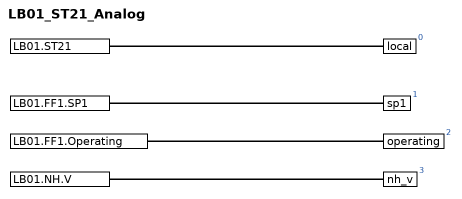
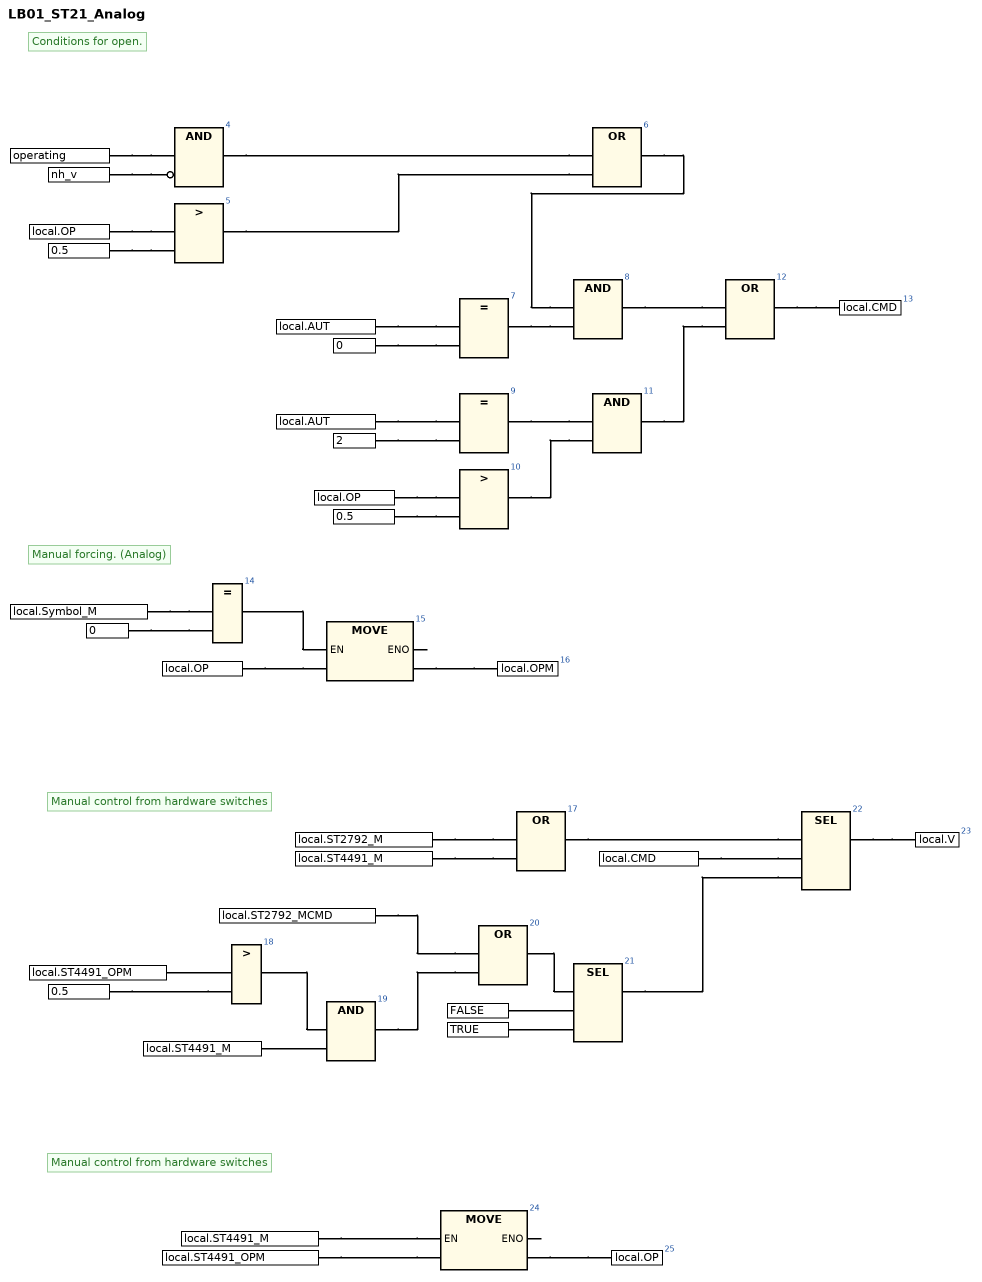
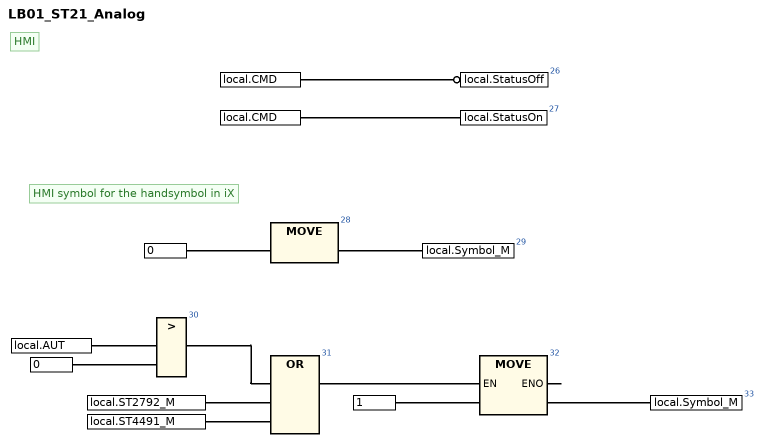
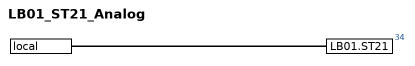
local := LB01.ST21;
sp1 := LB01.FF1.SP1;
operating := LB01.FF1.Operating;
nh_v := LB01.NH.V;
// Conditions for open.
local.CMD := (operating AND NOT nh_v OR local.OP > 0.5) AND local.AUT = 0 OR local.AUT = 2 AND local.OP > 0.5;
// Manual forcing. (Analog)
IF local.Symbol_M = 0 THEN _w1 := local.OP; END_IF
local.OPM := _w1;
// Manual control from hardware switches
local.V := SEL(local.ST2792_M OR local.ST4491_M, local.CMD, SEL(local.ST2792_MCMD OR local.ST4491_OPM > 0.5 AND local.ST4491_M, FALSE, TRUE));
// Manual control from hardware switches
IF local.ST4491_M THEN _w2 := local.ST4491_OPM; END_IF
local.OP := _w2;
// HMI
local.StatusOff := NOT local.CMD;
local.StatusOn := local.CMD;
// HMI symbol for the handsymbol in iX
local.Symbol_M := 0;
IF local.AUT > 0 OR local.ST2792_M OR local.ST4491_M THEN _w3 := 1; END_IF
local.Symbol_M := _w3;
LB01.ST21 := local;

END_PROGRAM

// Device/AREA1/B001/LB01/Fan/TF1/LB01_TF1_OneSpeed
PROGRAM LB01_TF1_OneSpeed
VAR
	local:strFan_Onespeed;
	_BE_Fan2:_BE_Fan_2;
	AlarmFbAl01: _BE_AlarmAckRequired;
	AlarmFbAl02: _BE_AlarmAckRequired;
	fb_OperationalTime: _BE_OperationalTime;
	ackAl01: BOOL;
	ackAl02: BOOL;
	fanGuardOk: BOOL;
END_VAR

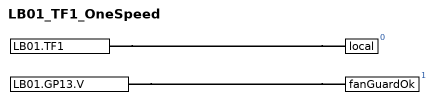
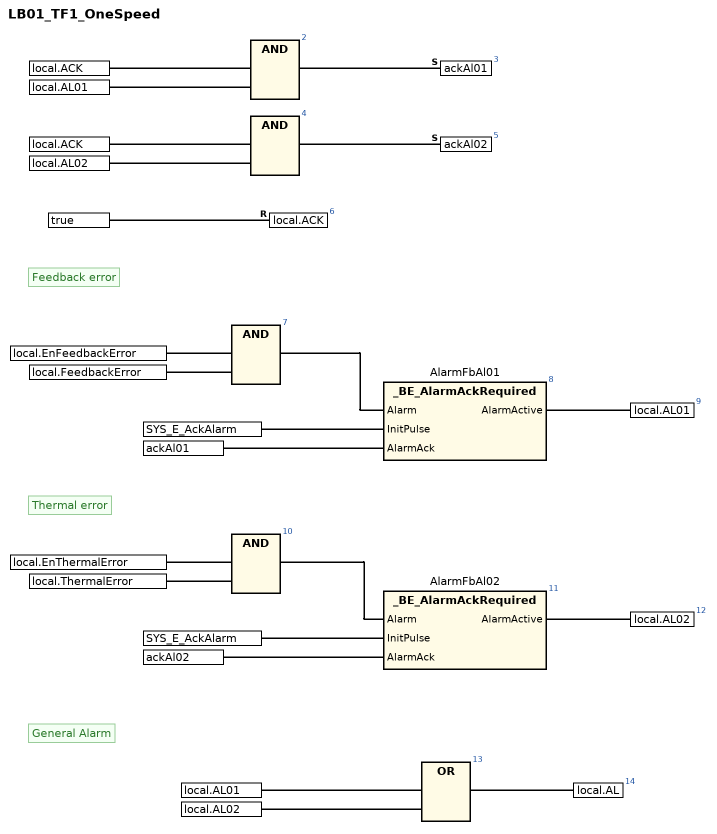
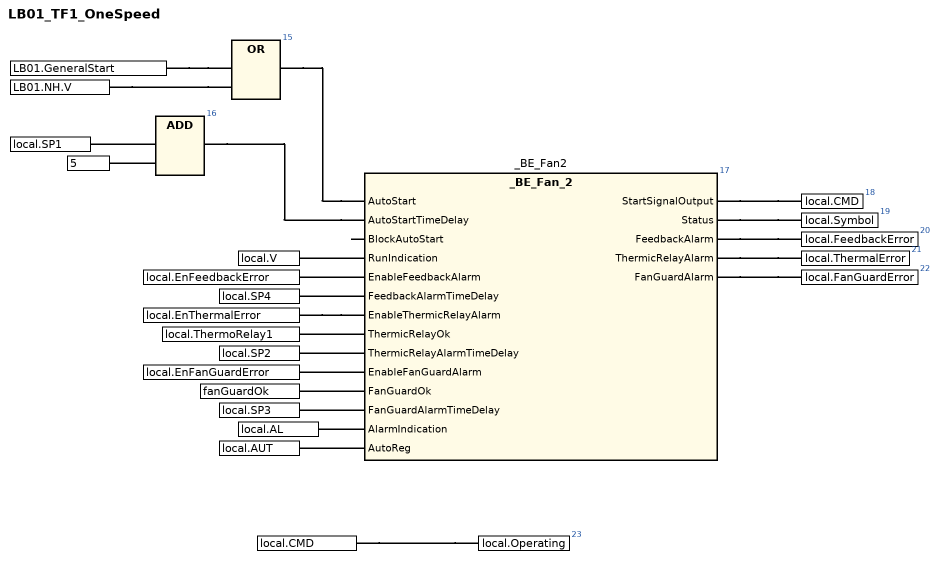
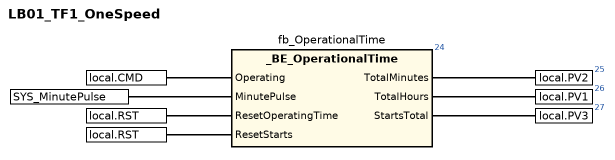
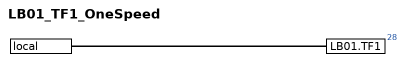
local := LB01.TF1;
fanGuardOk := LB01.GP13.V;
ackAl01 S= local.ACK AND local.AL01;
ackAl02 S= local.ACK AND local.AL02;
local.ACK R= true;
// Feedback error
AlarmFbAl01(
    Alarm := local.EnFeedbackError AND local.FeedbackError,
    InitPulse := SYS_E_AckAlarm,
    AlarmAck := ackAl01); // _BE_AlarmAckRequired
local.AL01 := AlarmFbAl01.AlarmActive;
// Thermal error
AlarmFbAl02(
    Alarm := local.EnThermalError AND local.ThermalError,
    InitPulse := SYS_E_AckAlarm,
    AlarmAck := ackAl02); // _BE_AlarmAckRequired
local.AL02 := AlarmFbAl02.AlarmActive;
// General Alarm
local.AL := local.AL01 OR local.AL02;
_BE_Fan2(
    AutoStart := LB01.GeneralStart OR LB01.NH.V,
    AutoStartTimeDelay := local.SP1 + 5,
    RunIndication := local.V,
    EnableFeedbackAlarm := local.EnFeedbackError,
    FeedbackAlarmTimeDelay := local.SP4,
    EnableThermicRelayAlarm := local.EnThermalError,
    ThermicRelayOk := local.ThermoRelay1,
    ThermicRelayAlarmTimeDelay := local.SP2,
    EnableFanGuardAlarm := local.EnFanGuardError,
    FanGuardOk := fanGuardOk,
    FanGuardAlarmTimeDelay := local.SP3,
    AlarmIndication := local.AL,
    AutoReg := local.AUT); // _BE_Fan_2
local.CMD := _BE_Fan2.StartSignalOutput;
local.Symbol := _BE_Fan2.Status;
local.FeedbackError := _BE_Fan2.FeedbackAlarm;
local.ThermalError := _BE_Fan2.ThermicRelayAlarm;
local.FanGuardError := _BE_Fan2.FanGuardAlarm;
local.Operating := local.CMD;
fb_OperationalTime(
    Operating := local.CMD,
    MinutePulse := SYS_MinutePulse,
    ResetOperatingTime := local.RST,
    ResetStarts := local.RST); // _BE_OperationalTime
local.PV2 := fb_OperationalTime.TotalMinutes;
local.PV1 := fb_OperationalTime.TotalHours;
local.PV3 := fb_OperationalTime.StartsTotal;
LB01.TF1 := local;

END_PROGRAM

// Device/AREA1/B001/LB01/Fan/TF1/LB01_TF1_TwoSpeed
PROGRAM LB01_TF1_TwoSpeed
VAR
	local:strFan_TwoSpeed;
	ControlTwoSpeed: _BE_FanTwoSpeed;
	AlarmFbAl03: _BE_AlarmAckRequired;
	AlarmFbAl04: _BE_AlarmAckRequired;
	AlarmFbAl05: _BE_AlarmAckRequired;
	AlarmFbAl06: _BE_AlarmAckRequired;
	ackAl03: BOOL;
	ackAl04: BOOL;
	ackAl05: BOOL;
	ackAl06: BOOL;
	fb_OperationalTime: _BE_OperationalTime;
	localV1: BOOL;
	localthermoRelay2: BOOL;
	fanGuardOk: BOOL;
END_VAR
VAR // added by the converter: edge detectors and wires of the graphical bodies
    _w1 : ANY;
END_VAR

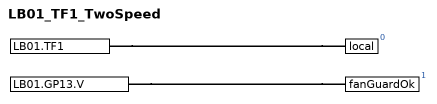
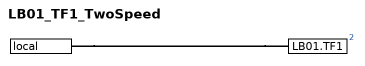
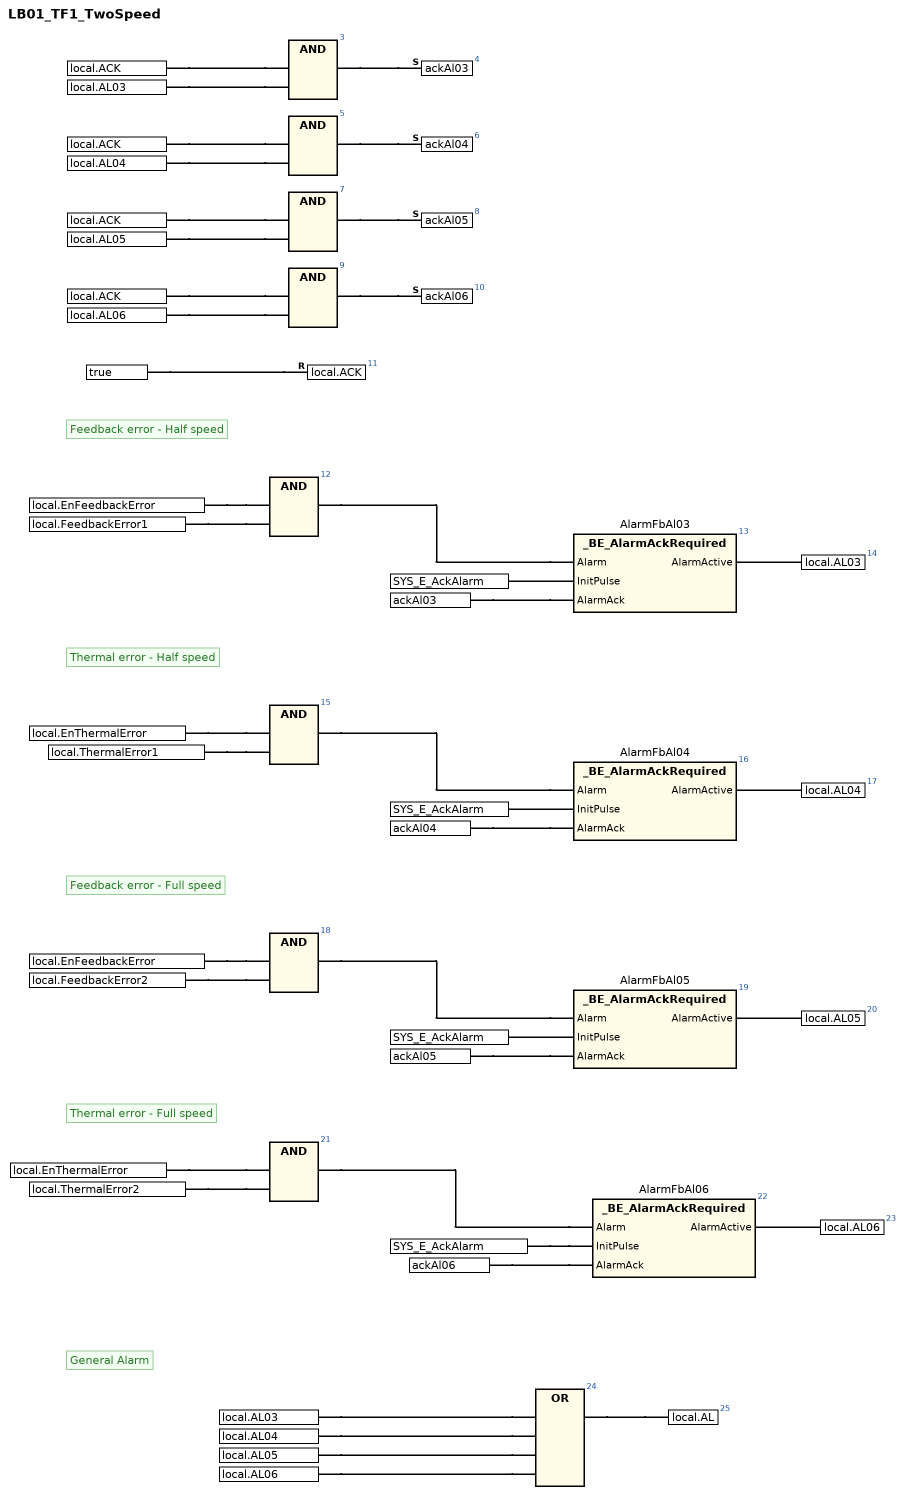
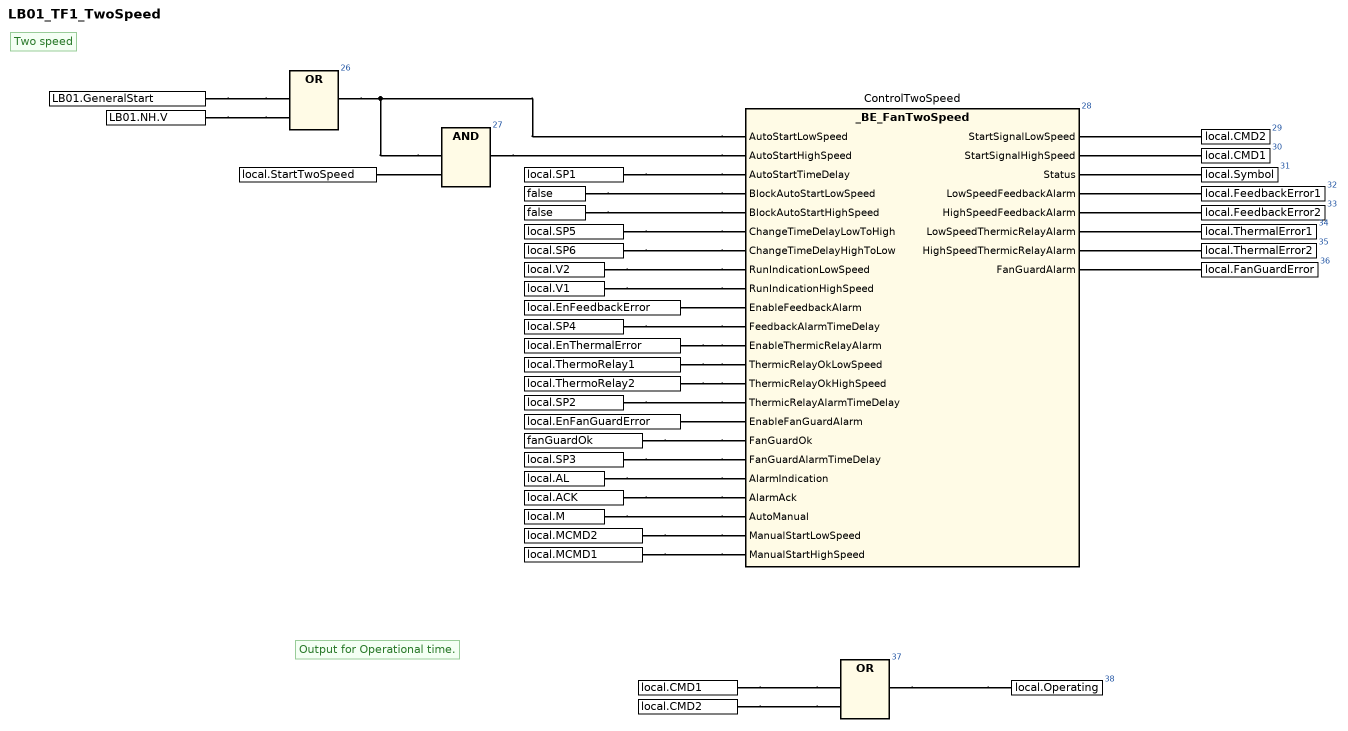
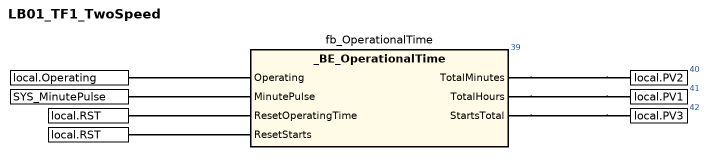
local := LB01.TF1;
fanGuardOk := LB01.GP13.V;
LB01.TF1 := local;
ackAl03 S= local.ACK AND local.AL03;
ackAl04 S= local.ACK AND local.AL04;
ackAl05 S= local.ACK AND local.AL05;
ackAl06 S= local.ACK AND local.AL06;
local.ACK R= true;
// Feedback error - Half speed
AlarmFbAl03(
    Alarm := local.EnFeedbackError AND local.FeedbackError1,
    InitPulse := SYS_E_AckAlarm,
    AlarmAck := ackAl03); // _BE_AlarmAckRequired
local.AL03 := AlarmFbAl03.AlarmActive;
// Thermal error - Half speed
AlarmFbAl04(
    Alarm := local.EnThermalError AND local.ThermalError1,
    InitPulse := SYS_E_AckAlarm,
    AlarmAck := ackAl04); // _BE_AlarmAckRequired
local.AL04 := AlarmFbAl04.AlarmActive;
// Feedback error - Full speed
AlarmFbAl05(
    Alarm := local.EnFeedbackError AND local.FeedbackError2,
    InitPulse := SYS_E_AckAlarm,
    AlarmAck := ackAl05); // _BE_AlarmAckRequired
local.AL05 := AlarmFbAl05.AlarmActive;
// Thermal error - Full speed
AlarmFbAl06(
    Alarm := local.EnThermalError AND local.ThermalError2,
    InitPulse := SYS_E_AckAlarm,
    AlarmAck := ackAl06); // _BE_AlarmAckRequired
local.AL06 := AlarmFbAl06.AlarmActive;
// General Alarm
local.AL := local.AL03 OR local.AL04 OR local.AL05 OR local.AL06;
// Two speed
_w1 := LB01.GeneralStart OR LB01.NH.V;
ControlTwoSpeed(
    AutoStartLowSpeed := _w1,
    AutoStartHighSpeed := _w1 AND local.StartTwoSpeed,
    AutoStartTimeDelay := local.SP1,
    BlockAutoStartLowSpeed := false,
    BlockAutoStartHighSpeed := false,
    ChangeTimeDelayLowToHigh := local.SP5,
    ChangeTimeDelayHighToLow := local.SP6,
    RunIndicationLowSpeed := local.V2,
    RunIndicationHighSpeed := local.V1,
    EnableFeedbackAlarm := local.EnFeedbackError,
    FeedbackAlarmTimeDelay := local.SP4,
    EnableThermicRelayAlarm := local.EnThermalError,
    ThermicRelayOkLowSpeed := local.ThermoRelay1,
    ThermicRelayOkHighSpeed := local.ThermoRelay2,
    ThermicRelayAlarmTimeDelay := local.SP2,
    EnableFanGuardAlarm := local.EnFanGuardError,
    FanGuardOk := fanGuardOk,
    FanGuardAlarmTimeDelay := local.SP3,
    AlarmIndication := local.AL,
    AlarmAck := local.ACK,
    AutoManual := local.M,
    ManualStartLowSpeed := local.MCMD2,
    ManualStartHighSpeed := local.MCMD1); // _BE_FanTwoSpeed
local.CMD2 := ControlTwoSpeed.StartSignalLowSpeed;
local.CMD1 := ControlTwoSpeed.StartSignalHighSpeed;
local.Symbol := ControlTwoSpeed.Status;
local.FeedbackError1 := ControlTwoSpeed.LowSpeedFeedbackAlarm;
local.FeedbackError2 := ControlTwoSpeed.HighSpeedFeedbackAlarm;
local.ThermalError1 := ControlTwoSpeed.LowSpeedThermicRelayAlarm;
local.ThermalError2 := ControlTwoSpeed.HighSpeedThermicRelayAlarm;
local.FanGuardError := ControlTwoSpeed.FanGuardAlarm;
// Output for Operational time.
local.Operating := local.CMD1 OR local.CMD2;
fb_OperationalTime(
    Operating := local.Operating,
    MinutePulse := SYS_MinutePulse,
    ResetOperatingTime := local.RST,
    ResetStarts := local.RST); // _BE_OperationalTime
local.PV2 := fb_OperationalTime.TotalMinutes;
local.PV1 := fb_OperationalTime.TotalHours;
local.PV3 := fb_OperationalTime.StartsTotal;

END_PROGRAM

// Device/AREA1/B001/LB01/Function/LB01_Function_OutsideCompensation
PROGRAM LB01_Function_OutsideCompensation
VAR
	FbOutsideCompensation: _BE_OutCompSevenSetPoint;
END_VAR

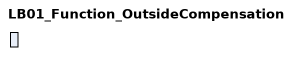
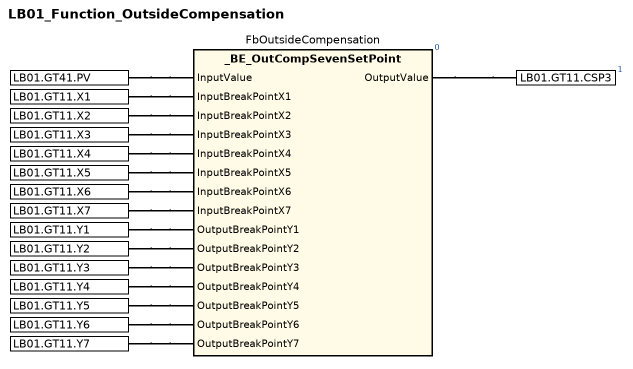
FbOutsideCompensation(
    InputValue := LB01.GT41.PV,
    InputBreakPointX1 := LB01.GT11.X1,
    InputBreakPointX2 := LB01.GT11.X2,
    InputBreakPointX3 := LB01.GT11.X3,
    InputBreakPointX4 := LB01.GT11.X4,
    InputBreakPointX5 := LB01.GT11.X5,
    InputBreakPointX6 := LB01.GT11.X6,
    InputBreakPointX7 := LB01.GT11.X7,
    OutputBreakPointY1 := LB01.GT11.Y1,
    OutputBreakPointY2 := LB01.GT11.Y2,
    OutputBreakPointY3 := LB01.GT11.Y3,
    OutputBreakPointY4 := LB01.GT11.Y4,
    OutputBreakPointY5 := LB01.GT11.Y5,
    OutputBreakPointY6 := LB01.GT11.Y6,
    OutputBreakPointY7 := LB01.GT11.Y7); // _BE_OutCompSevenSetPoint
LB01.GT11.CSP3 := FbOutsideCompensation.OutputValue;

END_PROGRAM

// Device/AREA1/B001/LB01/Function/LB01_Function_EfficiencySupplyAir
PROGRAM LB01_Function_EfficiencySupplyAir
VAR
	FbEfficiency: _BE_RecoveryEfficiencyExtractAir;
	gt_Min: TON;
	AlarmAcknowledge01: _BE_AlarmAckRemote;
END_VAR

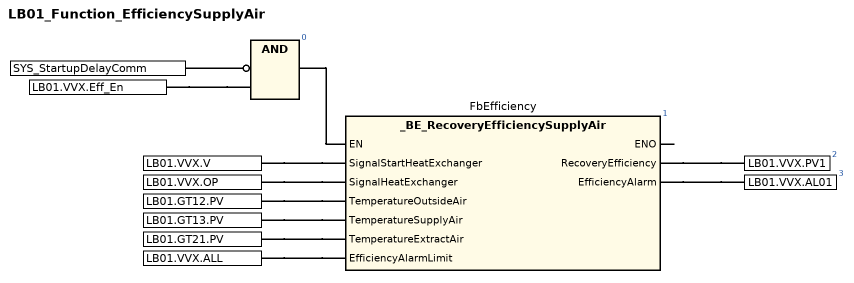
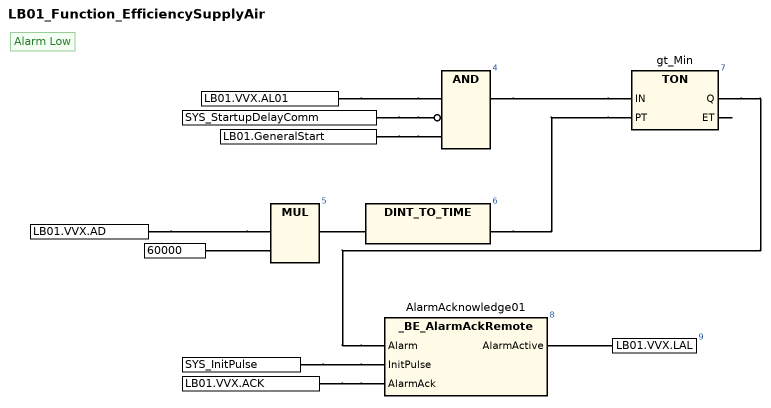
IF NOT SYS_StartupDelayComm AND LB01.VVX.Eff_En THEN
    FbEfficiency(
        SignalStartHeatExchanger := LB01.VVX.V,
        SignalHeatExchanger := LB01.VVX.OP,
        TemperatureOutsideAir := LB01.GT12.PV,
        TemperatureSupplyAir := LB01.GT13.PV,
        TemperatureExtractAir := LB01.GT21.PV,
        EfficiencyAlarmLimit := LB01.VVX.ALL); // _BE_RecoveryEfficiencySupplyAir
END_IF
LB01.VVX.PV1 := FbEfficiency.RecoveryEfficiency;
LB01.VVX.AL01 := FbEfficiency.EfficiencyAlarm;
// Alarm Low
gt_Min(IN := LB01.VVX.AL01 AND NOT SYS_StartupDelayComm AND LB01.GeneralStart, PT := DINT_TO_TIME(LB01.VVX.AD * 60000)); // TON
AlarmAcknowledge01(Alarm := gt_Min.Q, InitPulse := SYS_InitPulse, AlarmAck := LB01.VVX.ACK); // _BE_AlarmAckRemote
LB01.VVX.LAL := AlarmAcknowledge01.AlarmActive;

END_PROGRAM

// Device/AREA1/B001/LB01/HeatExchanger/LB01_HeatExchanger_Cross
PROGRAM LB01_HeatExchanger_Cross
VAR
	local:strHeatExchanger_Cross;
	inputValue: LREAL;
	FbAnalogOverride: _BE_AnalogueOverride;
	inputAlarm: BOOL;
	nh_v: BOOL;
	FbTofmin: TOF;
END_VAR
VAR // added by the converter: edge detectors and wires of the graphical bodies
    _w1, _w3, _w5, _w6, _w7 : ANY;
    _w2, _w4 : BOOL;
END_VAR

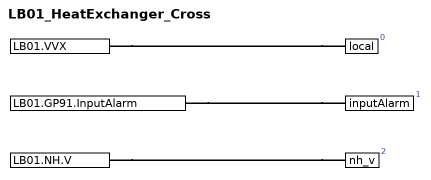
